// TIA Portal V16 export
// export: Created 2022-11-17T11:55:21.4040062Z, ExportSetting WithDefaults, DisplayName Totally Integrated Automation Portal, DisplayVersion V16 Update 6, DisplayName TIA Portal Version Control Interface, DisplayVersion V16 Update 2, DisplayName TIA Portal Openness, DisplayVersion V16 Update 6, DisplayName SINAMICS Startdrive Advanced, DisplayVersion V16 Update 5, DisplayName SINAMICS Startdrive G130, G150, S120, S150, SINAMICS MV, S210, DisplayVersion V16 Update 5, DisplayName SINAMICS Startdrive G110M, G120, G120C, G120D, G120P, G115D, DisplayVersion V16 Update 5, DisplayName STEP 7 Professional, DisplayVersion V16 Update 6, DisplayName STEP 7 Safety, DisplayVersion V16, DisplayName WinCC Advanced, DisplayVersion V16 Update 6
FUNCTION "FC105_GreyBarReset" : Void   // FC105, LAD
TITLE = Reset grey bar program data
{ S7_Optimized_Access := 'TRUE' }
VERSION : 0.1
// stored: AutoNumber false, IsIECCheckEnabled false, SetENOAutomatically false, UDAEnableTagReadback false
BEGIN

REGION Network 1: Reset grey bar program data
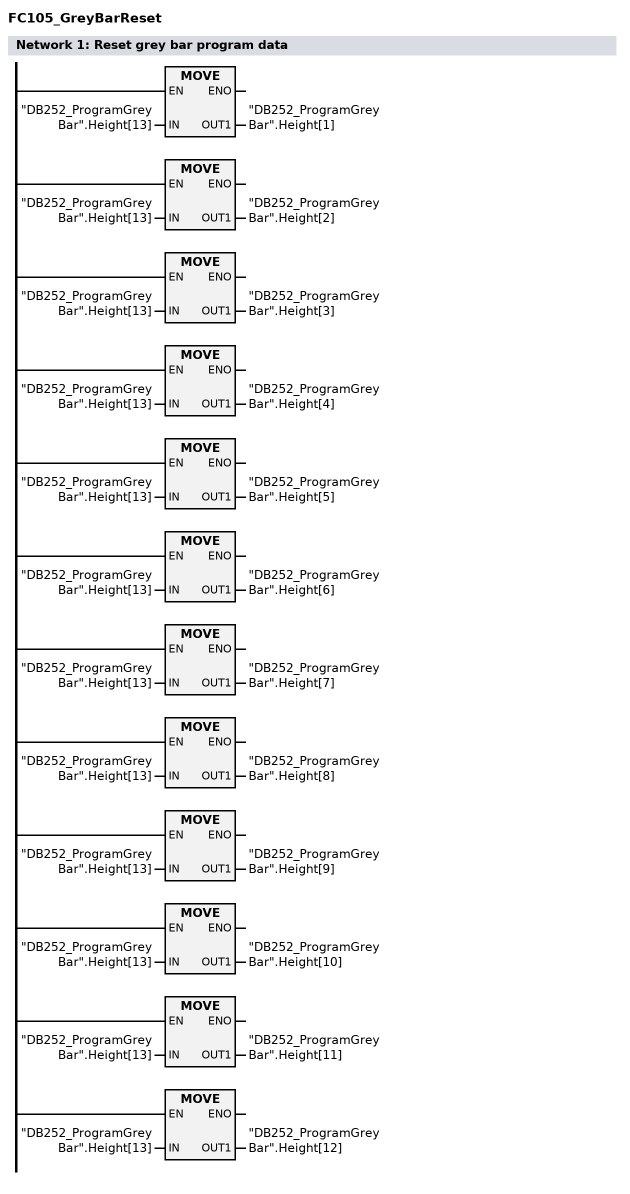
   RUNG wire#powerrail
      { S7_GenerateENO := "TRUE" } Move(in := "DB252_ProgramGreyBar".Height[13], out1 => "DB252_ProgramGreyBar".Height[1])
   END_RUNG
   RUNG wire#powerrail
      { S7_GenerateENO := "TRUE" } Move(in := "DB252_ProgramGreyBar".Height[13], out1 => "DB252_ProgramGreyBar".Height[2])
   END_RUNG
   RUNG wire#powerrail
      { S7_GenerateENO := "TRUE" } Move(in := "DB252_ProgramGreyBar".Height[13], out1 => "DB252_ProgramGreyBar".Height[3])
   END_RUNG
   RUNG wire#powerrail
      { S7_GenerateENO := "TRUE" } Move(in := "DB252_ProgramGreyBar".Height[13], out1 => "DB252_ProgramGreyBar".Height[4])
   END_RUNG
   RUNG wire#powerrail
      { S7_GenerateENO := "TRUE" } Move(in := "DB252_ProgramGreyBar".Height[13], out1 => "DB252_ProgramGreyBar".Height[5])
   END_RUNG
   RUNG wire#powerrail
      { S7_GenerateENO := "TRUE" } Move(in := "DB252_ProgramGreyBar".Height[13], out1 => "DB252_ProgramGreyBar".Height[6])
   END_RUNG
   RUNG wire#powerrail
      { S7_GenerateENO := "TRUE" } Move(in := "DB252_ProgramGreyBar".Height[13], out1 => "DB252_ProgramGreyBar".Height[7])
   END_RUNG
   RUNG wire#powerrail
      { S7_GenerateENO := "TRUE" } Move(in := "DB252_ProgramGreyBar".Height[13], out1 => "DB252_ProgramGreyBar".Height[8])
   END_RUNG
   RUNG wire#powerrail
      { S7_GenerateENO := "TRUE" } Move(in := "DB252_ProgramGreyBar".Height[13], out1 => "DB252_ProgramGreyBar".Height[9])
   END_RUNG
   RUNG wire#powerrail
      { S7_GenerateENO := "TRUE" } Move(in := "DB252_ProgramGreyBar".Height[13], out1 => "DB252_ProgramGreyBar".Height[10])
   END_RUNG
   RUNG wire#powerrail
      { S7_GenerateENO := "TRUE" } Move(in := "DB252_ProgramGreyBar".Height[13], out1 => "DB252_ProgramGreyBar".Height[11])
   END_RUNG
   RUNG wire#powerrail
      { S7_GenerateENO := "TRUE" } Move(in := "DB252_ProgramGreyBar".Height[13], out1 => "DB252_ProgramGreyBar".Height[12])
   END_RUNG
   // the same network as SCL:
   "DB252_ProgramGreyBar".Height[1] := "DB252_ProgramGreyBar".Height[13];
   "DB252_ProgramGreyBar".Height[2] := "DB252_ProgramGreyBar".Height[13];
   "DB252_ProgramGreyBar".Height[3] := "DB252_ProgramGreyBar".Height[13];
   "DB252_ProgramGreyBar".Height[4] := "DB252_ProgramGreyBar".Height[13];
   "DB252_ProgramGreyBar".Height[5] := "DB252_ProgramGreyBar".Height[13];
   "DB252_ProgramGreyBar".Height[6] := "DB252_ProgramGreyBar".Height[13];
   "DB252_ProgramGreyBar".Height[7] := "DB252_ProgramGreyBar".Height[13];
   "DB252_ProgramGreyBar".Height[8] := "DB252_ProgramGreyBar".Height[13];
   "DB252_ProgramGreyBar".Height[9] := "DB252_ProgramGreyBar".Height[13];
   "DB252_ProgramGreyBar".Height[10] := "DB252_ProgramGreyBar".Height[13];
   "DB252_ProgramGreyBar".Height[11] := "DB252_ProgramGreyBar".Height[13];
   "DB252_ProgramGreyBar".Height[12] := "DB252_ProgramGreyBar".Height[13];
END_REGION
END_FUNCTION
